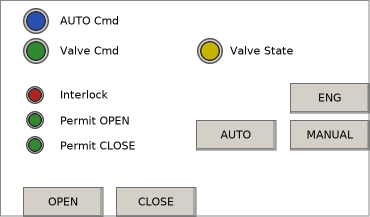
VISUALIZATION GUI_TEMPLATE_ACTUATOR_ENG  // 370x217
VAR_IN_OUT
	m_Cmd:		FB_CRYO_ACTUATOR_CMD;
	m_Valve:	FB_CRYO_VALVE_CTRL;
END_VAR
    Lamp1 (25,85 20x20), variable: m_Cmd.in_bInterlock, style: Lamp-Lamp1-Red
    Lamp1 (25,110 20x20), variable: m_Cmd.bPermitOn, style: Lamp-Lamp1-Green
    Lamp1 (25,135 20x20), variable: m_Cmd.bPermitOff, style: Lamp-Lamp1-Green
    Rectangle (57,80 83x30), "Interlock"
    Rectangle (57,106 83x30), "Permit OPEN"
    Rectangle (57,131 83x30), "Permit CLOSE"
    Button (23,187 80x30), "OPEN", colour toggle: (m_Cmd.bPermitOn AND NOT m_Cmd.bAutoMode) OR m_Cmd.bEngMode, input disabled if: m_Cmd.bDisableBtnOn
        OnMouseClick: execute { m_Cmd.bManualCmd := TRUE; m_Cmd.bManualExecute := TRUE; }
    Lamp1 (21,36 30x30), tooltip "Actual Valve command", variable: m_Cmd.out_bEnable, style: Lamp-Lamp1-Green
    Rectangle (57,36 83x30), "Valve Cmd"
    Button (196,120 80x30), "AUTO", colour toggle: m_Cmd.bAutoMode, input disabled if: m_Cmd.bAutoMode OR m_Cmd.bEngMode
        OnMouseClick: execute { m_Cmd.bAutoMode := TRUE; }
    Button (290,120 80x30), "MANUAL", colour toggle: NOT m_Cmd.bAutoMode, input disabled if: NOT m_Cmd.bAutoMode AND NOT m_Cmd.bEngMode
        OnMouseClick: execute { m_Cmd.bAutoMode := FALSE; }
    Button (116,187 80x30), "CLOSE", colour toggle: (m_Cmd.bPermitOff AND NOT m_Cmd.bAutoMode) OR m_Cmd.bEngMode, input disabled if: m_Cmd.bDisableBtnOff
        OnMouseClick: execute { m_Cmd.bManualCmd := FALSE; m_Cmd.bManualExecute := TRUE; }
    Button (290,83 80x30), "ENG", tooltip "Engineering / Commissioning Mode", colour toggle: m_Cmd.bEngMode, input disabled if: m_Cmd.bAutoMode
        toggle m_Cmd.bEngMode
    Lamp1 (21,6 30x30), tooltip "Command coming from the Control System", variable: m_Cmd.in_bEnable, style: Lamp-Lamp1-Blue
    Rectangle (57,6 83x30), "AUTO Cmd"
    Lamp1 (195,36 30x30), tooltip "Valve state: ON=OPEN, OFF=CLOSED", variable: m_Valve.stat.bActON, style: Lamp-Lamp1-Yellow
    Rectangle (227,36 83x30), "Valve State"
END_VISUALIZATION

(* stored: Version 1.1.0.1, ProductVersion 3.1.4024.12
   Visu GUI_TEMPLATE_ACTUATOR_ENG: Id {5cac297a-c120-46a4-8fe5-e7e7dbf68e0c} *)
